{attribute wpf [Container(Layout.Stack)]}
TYPE LayoutStackStruct EXTENDS VariousTypesStruct :
STRUCT
END_STRUCT
END_TYPE

(* stored: Version 1.1.0.1, ProductVersion 3.1.4024.9
   DUT LayoutStackStruct: Id {ef44e3d6-b837-4bb4-89da-d5be138072ef} *)
